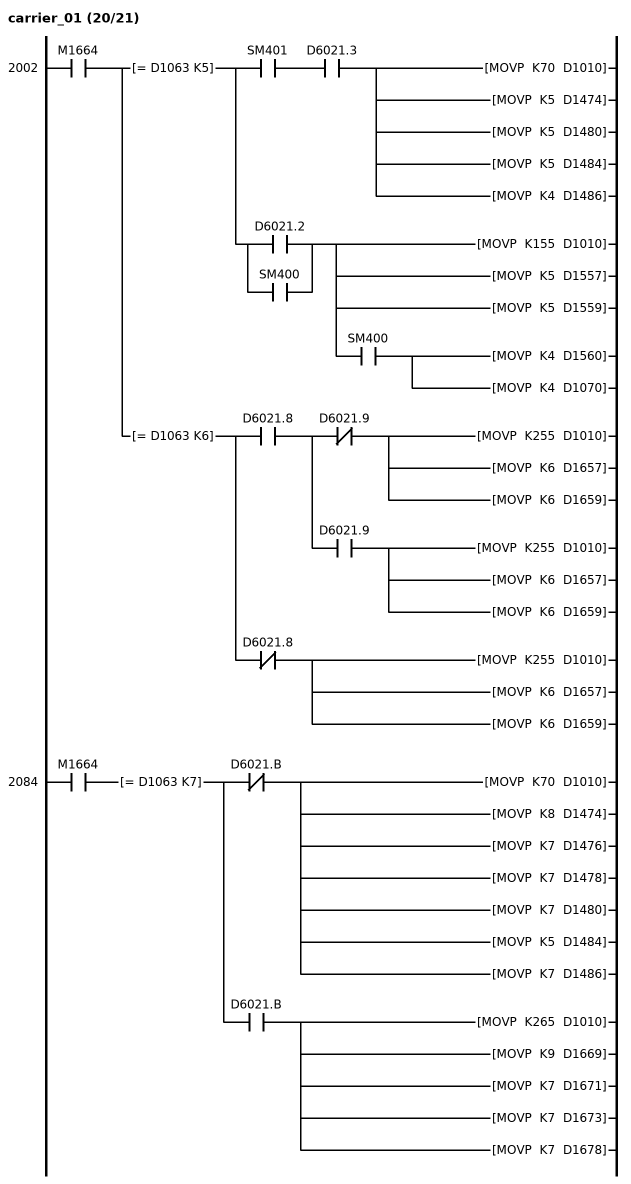
[picture p48: ladder of carrier_01, rungs at steps 2002 to 2084]
2002  LD      M1664
      MPS
      AND=    D1063 K5
      MPS
      AND     SM401
      AND     D6021.3
      MOVP    K70 D1010
      MOVP    K5 D1474
      MOVP    K5 D1480
      MOVP    K5 D1484
      MOVP    K4 D1486
      MPP
      LD      D6021.2
      OR      SM400
      ANB
      MOVP    K155 D1010
      MOVP    K5 D1557
      MOVP    K5 D1559
      AND     SM400
      MOVP    K4 D1560
      MOVP    K4 D1070
      MPP
      AND=    D1063 K6
      MPS
      AND     D6021.8
      MPS
      ANI     D6021.9
      MOVP    K255 D1010
      MOVP    K6 D1657
      MOVP    K6 D1659
      MPP
      AND     D6021.9
      MOVP    K255 D1010
      MOVP    K6 D1657
      MOVP    K6 D1659
      MPP
      ANI     D6021.8
      MOVP    K255 D1010
      MOVP    K6 D1657
      MOVP    K6 D1659
2084  LD      M1664
      AND=    D1063 K7
      MPS
      ANI     D6021.B
      MOVP    K70 D1010
      MOVP    K8 D1474
      MOVP    K7 D1476
      MOVP    K7 D1478
      MOVP    K7 D1480
      MOVP    K5 D1484
      MOVP    K7 D1486
      MPP
      AND     D6021.B
      MOVP    K265 D1010
      MOVP    K9 D1669
      MOVP    K7 D1671
      MOVP    K7 D1673
      MOVP    K7 D1678
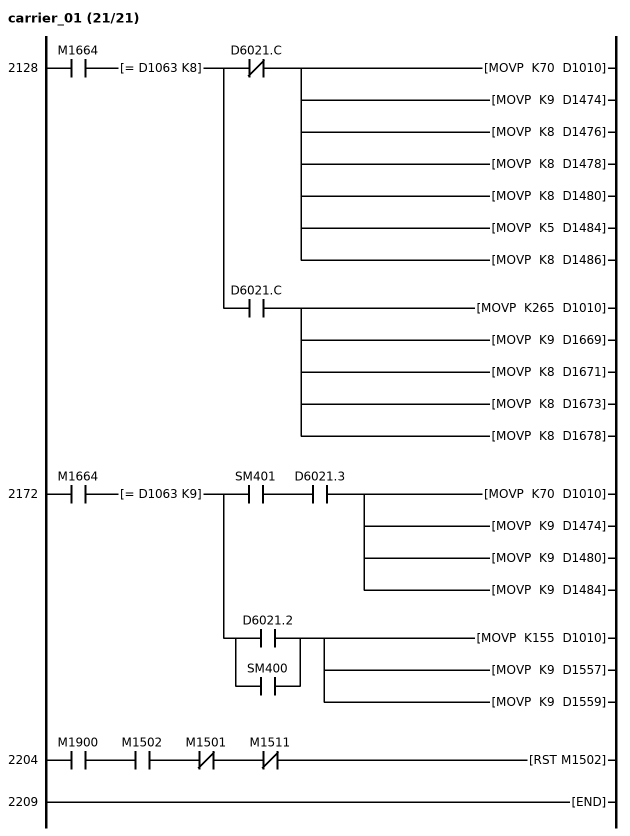
2128  LD      M1664
      AND=    D1063 K8
      MPS
      ANI     D6021.C
      MOVP    K70 D1010
      MOVP    K9 D1474
      MOVP    K8 D1476
      MOVP    K8 D1478
      MOVP    K8 D1480
      MOVP    K5 D1484
      MOVP    K8 D1486
      MPP
      AND     D6021.C
      MOVP    K265 D1010
      MOVP    K9 D1669
      MOVP    K8 D1671
      MOVP    K8 D1673
      MOVP    K8 D1678
2172  LD      M1664
      AND=    D1063 K9
      MPS
      AND     SM401
      AND     D6021.3
      MOVP    K70 D1010
      MOVP    K9 D1474
      MOVP    K9 D1480
      MOVP    K9 D1484
      MPP
      LD      D6021.2
      OR      SM400
      ANB
      MOVP    K155 D1010
      MOVP    K9 D1557
      MOVP    K9 D1559
2204  LD      M1900
      AND     M1502
      ANI     M1501
      ANI     M1511
      RST     M1502
2209  END
END_PROGRAM

PROGRAM carrier_02
VAR
  c_comm_2 : c_comm_2;
END_VAR
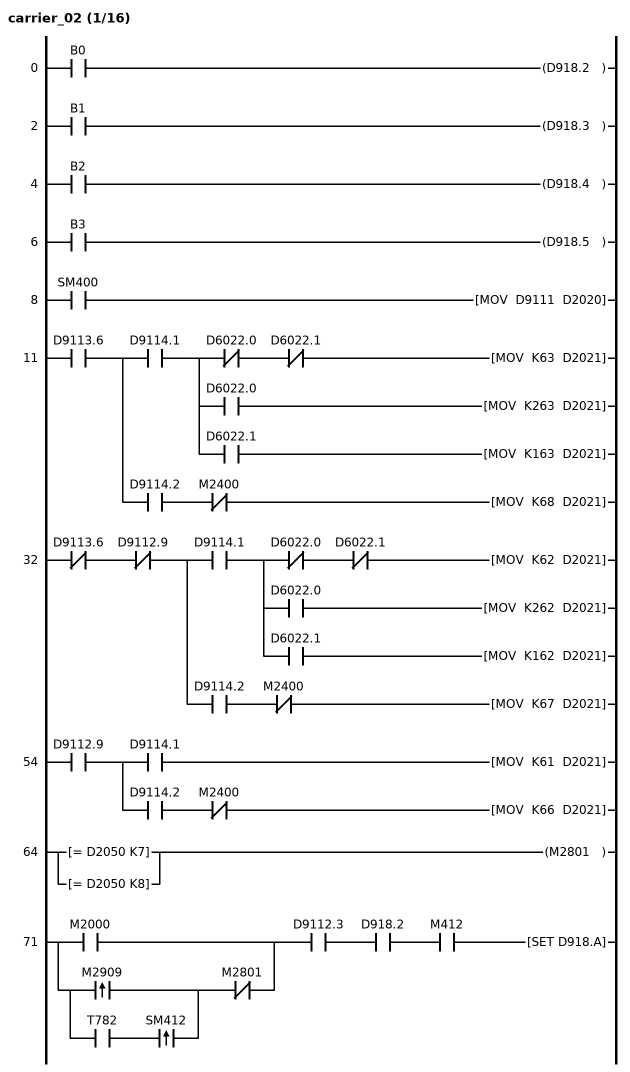
0     LD      B0
      OUT     D918.2
2     LD      B1
      OUT     D918.3
4     LD      B2
      OUT     D918.4
6     LD      B3
      OUT     D918.5
8     LD      SM400
      MOV     D9111 D2020
11    LD      D9113.6
      MPS
      AND     D9114.1
      MPS
      ANI     D6022.0
      ANI     D6022.1
      MOV     K63 D2021
      MRD
      AND     D6022.0
      MOV     K263 D2021
      MPP
      AND     D6022.1
      MOV     K163 D2021
      MPP
      AND     D9114.2
      ANI     M2400
      MOV     K68 D2021
32    LDI     D9113.6
      ANI     D9112.9
      MPS
      AND     D9114.1
      MPS
      ANI     D6022.0
      ANI     D6022.1
      MOV     K62 D2021
      MRD
      AND     D6022.0
      MOV     K262 D2021
      MPP
      AND     D6022.1
      MOV     K162 D2021
      MPP
      AND     D9114.2
      ANI     M2400
      MOV     K67 D2021
54    LD      D9112.9
      MPS
      AND     D9114.1
      MOV     K61 D2021
      MPP
      AND     D9114.2
      ANI     M2400
      MOV     K66 D2021
64    LD=     D2050 K7
      OR=     D2050 K8
      OUT     M2801
71    LD      M2000
      LDP     M2909
      LD      T782
      ANDP    SM412
      ORB
      ANI     M2801
      ORB
      AND     D9112.3
      AND     D918.2
      AND     M412
      SET     D918.A
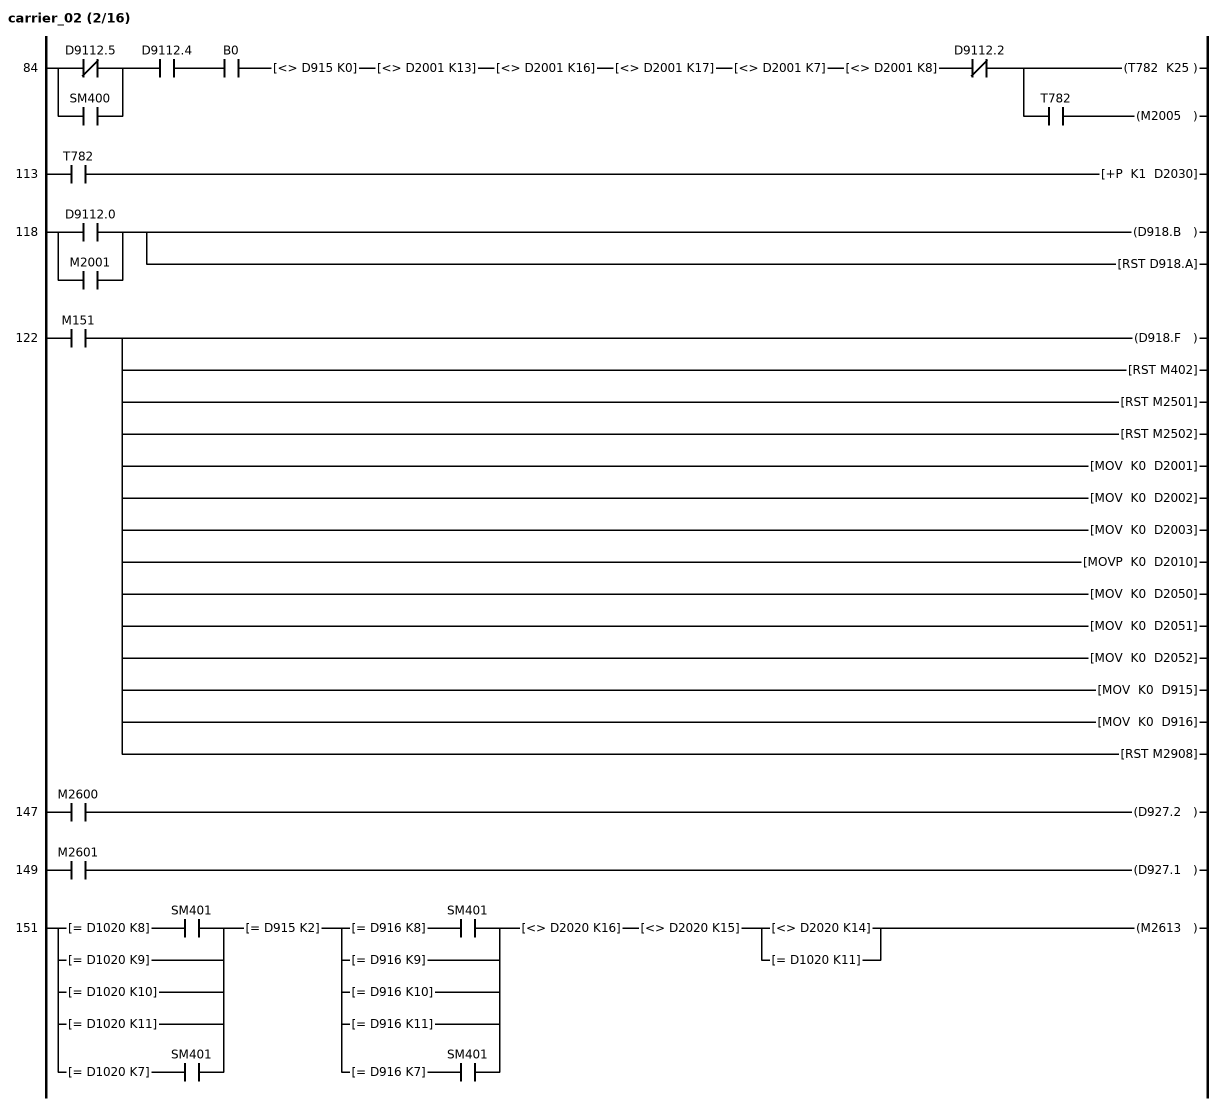
84    LDI     D9112.5
      OR      SM400
      AND     D9112.4
      AND     B0
      AND<>   D915 K0
      AND<>   D2001 K13
      AND<>   D2001 K16
      AND<>   D2001 K17
      AND<>   D2001 K7
      AND<>   D2001 K8
      ANI     D9112.2
      OUT     T782 K25
      AND     T782
      OUT     M2005
113   LD      T782
      +P      K1 D2030
118   LD      D9112.0
      OR      M2001
      OUT     D918.B
      RST     D918.A
122   LD      M151
      OUT     D918.F
      RST     M402
      RST     M2501
      RST     M2502
      MOV     K0 D2001
      MOV     K0 D2002
      MOV     K0 D2003
      MOVP    K0 D2010
      MOV     K0 D2050
      MOV     K0 D2051
      MOV     K0 D2052
      MOV     K0 D915
      MOV     K0 D916
      RST     M2908
147   LD      M2600
      OUT     D927.2
149   LD      M2601
      OUT     D927.1
151   LD=     D1020 K8
      AND     SM401
      OR=     D1020 K9
      OR=     D1020 K10
      OR=     D1020 K11
      LD=     D1020 K7
      AND     SM401
      ORB
      AND=    D915 K2
      LD=     D916 K8
      AND     SM401
      OR=     D916 K9
      OR=     D916 K10
      OR=     D916 K11
      LD=     D916 K7
      AND     SM401
      ORB
      ANB
      AND<>   D2020 K16
      AND<>   D2020 K15
      LD<>    D2020 K14
      OR=     D1020 K11
      ANB
      OUT     M2613
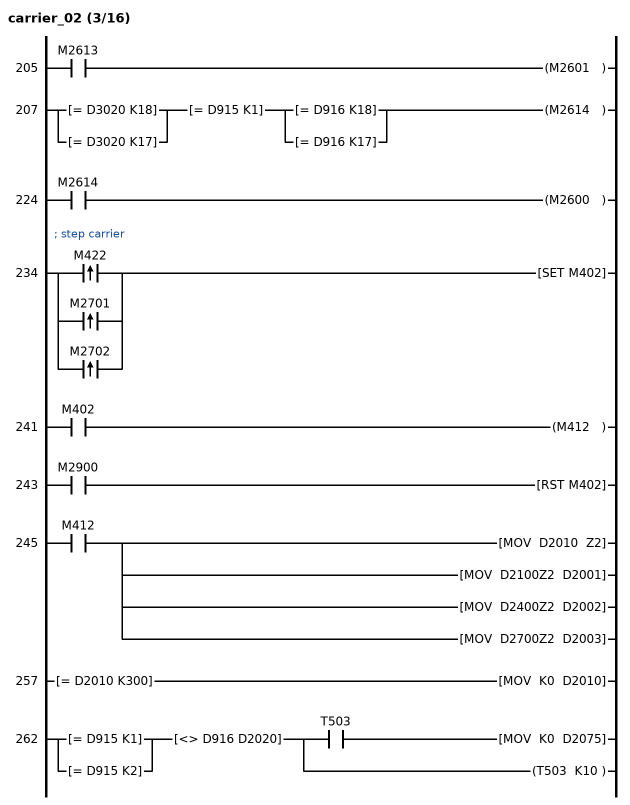
205   LD      M2613
      OUT     M2601
207   LD=     D3020 K18
      OR=     D3020 K17
      AND=    D915 K1
      LD=     D916 K18
      OR=     D916 K17
      ANB
      OUT     M2614
224   LD      M2614
      OUT     M2600
; step carrier
234   LDP     M422
      ORP     M2701
      ORP     M2702
      SET     M402
241   LD      M402
      OUT     M412
243   LD      M2900
      RST     M402
245   LD      M412
      MOV     D2010 Z2
      MOV     D2100Z2 D2001
      MOV     D2400Z2 D2002
      MOV     D2700Z2 D2003
257   LD=     D2010 K300
      MOV     K0 D2010
262   LD=     D915 K1
      OR=     D915 K2
      AND<>   D916 D2020
      MPS
      AND     T503
      MOV     K0 D2075
      MPP
      OUT     T503 K10
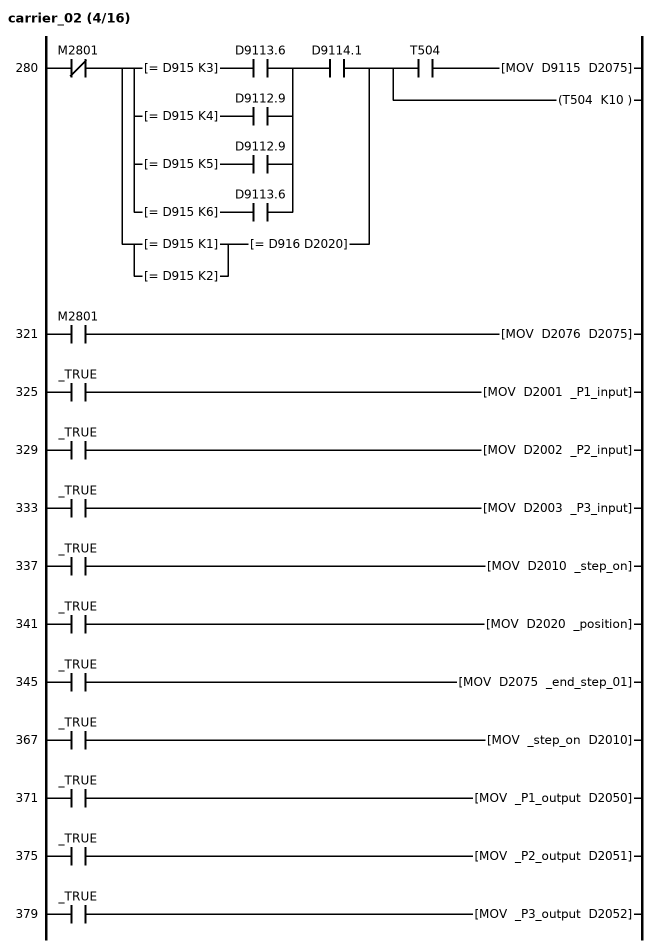
280   LDI     M2801
      LD=     D915 K3
      AND     D9113.6
      LD=     D915 K4
      AND     D9112.9
      ORB
      LD=     D915 K5
      AND     D9112.9
      ORB
      LD=     D915 K6
      AND     D9113.6
      ORB
      AND     D9114.1
      LD=     D915 K1
      OR=     D915 K2
      AND=    D916 D2020
      ORB
      ANB
      MPS
      AND     T504
      MOV     D9115 D2075
      MPP
      OUT     T504 K10
321   LD      M2801
      MOV     D2076 D2075
; FB BLK START c_comm_2(c_comm_2)
325   LD      _TRUE
      MOV     D2001 _P1_input
329   LD      _TRUE
      MOV     D2002 _P2_input
333   LD      _TRUE
      MOV     D2003 _P3_input
337   LD      _TRUE
      MOV     D2010 _step_on
341   LD      _TRUE
      MOV     D2020 _position
345   LD      _TRUE
      MOV     D2075 _end_step_01
; FB START
; FB_NAME c_comm_2
; INSTANCE_NAME c_comm_2
; FB IN_W:P1_input
; FB OUT_step_on:W
; FB IN_W:P2_input
; FB OUT_P1_output:W
; FB IN_W:P3_input
; FB OUT_P2_output:W
; FB IN_W:step_on
; FB OUT_P3_output:W
; FB IN_W:position
; FB OUT_end_step_01:W
; FB IN_W:end_step_01
; FB OUT_end_signal:B
; FB OUT_next_signal:B
; FB OUT_punch:B
; FB END
367   LD      _TRUE
      MOV     _step_on D2010
371   LD      _TRUE
      MOV     _P1_output D2050
375   LD      _TRUE
      MOV     _P2_output D2051
379   LD      _TRUE
      MOV     _P3_output D2052
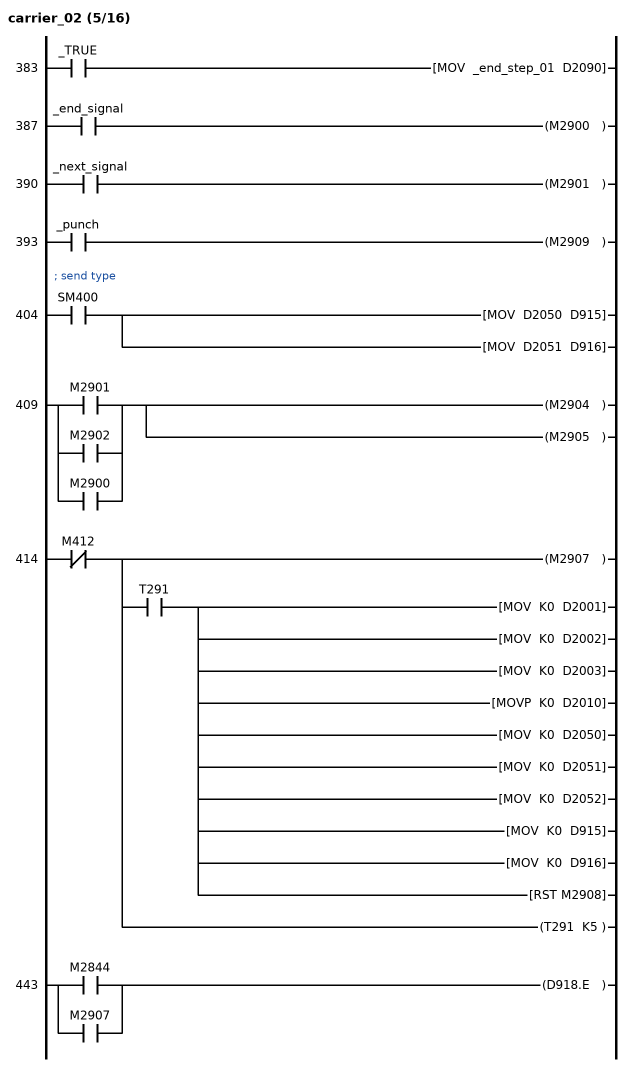
383   LD      _TRUE
      MOV     _end_step_01 D2090
387   LD      _end_signal
      OUT     M2900
390   LD      _next_signal
      OUT     M2901
393   LD      _punch
      OUT     M2909
; FB BLK END
; send type
404   LD      SM400
      MOV     D2050 D915
      MOV     D2051 D916
409   LD      M2901
      OR      M2902
      OR      M2900
      OUT     M2904
      OUT     M2905
414   LDI     M412
      OUT     M2907
      MPS
      AND     T291
      MOV     K0 D2001
      MOV     K0 D2002
      MOV     K0 D2003
      MOVP    K0 D2010
      MOV     K0 D2050
      MOV     K0 D2051
      MOV     K0 D2052
      MOV     K0 D915
      MOV     K0 D916
      RST     M2908
      MPP
      OUT     T291 K5
443   LD      M2844
      OR      M2907
      OUT     D918.E
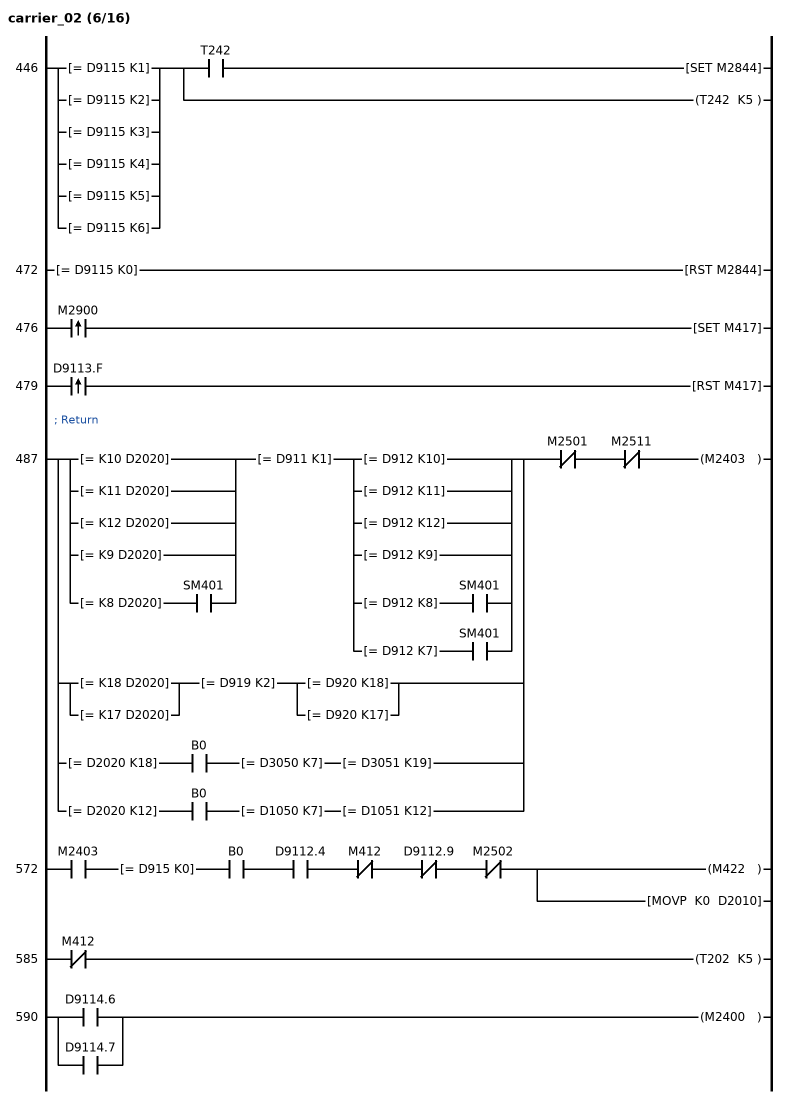
446   LD=     D9115 K1
      OR=     D9115 K2
      OR=     D9115 K3
      OR=     D9115 K4
      OR=     D9115 K5
      OR=     D9115 K6
      MPS
      AND     T242
      SET     M2844
      MPP
      OUT     T242 K5
472   LD=     D9115 K0
      RST     M2844
476   LDP     M2900
      SET     M417
479   LDP     D9113.F
      RST     M417
; Return
487   LD=     K10 D2020
      OR=     K11 D2020
      OR=     K12 D2020
      OR=     K9 D2020
      LD=     K8 D2020
      AND     SM401
      ORB
      AND=    D911 K1
      LD=     D912 K10
      OR=     D912 K11
      OR=     D912 K12
      OR=     D912 K9
      LD=     D912 K8
      AND     SM401
      ORB
      LD=     D912 K7
      AND     SM401
      ORB
      ANB
      LD=     K18 D2020
      OR=     K17 D2020
      AND=    D919 K2
      LD=     D920 K18
      OR=     D920 K17
      ANB
      ORB
      LD=     D2020 K18
      AND     B0
      AND=    D3050 K7
      AND=    D3051 K19
      ORB
      LD=     D2020 K12
      AND     B0
      AND=    D1050 K7
      AND=    D1051 K12
      ORB
      ANI     M2501
      ANI     M2511
      OUT     M2403
572   LD      M2403
      AND=    D915 K0
      AND     B0
      AND     D9112.4
      ANI     M412
      ANI     D9112.9
      ANI     M2502
      OUT     M422
      MOVP    K0 D2010
585   LDI     M412
      OUT     T202 K5
590   LD      D9114.6
      OR      D9114.7
      OUT     M2400
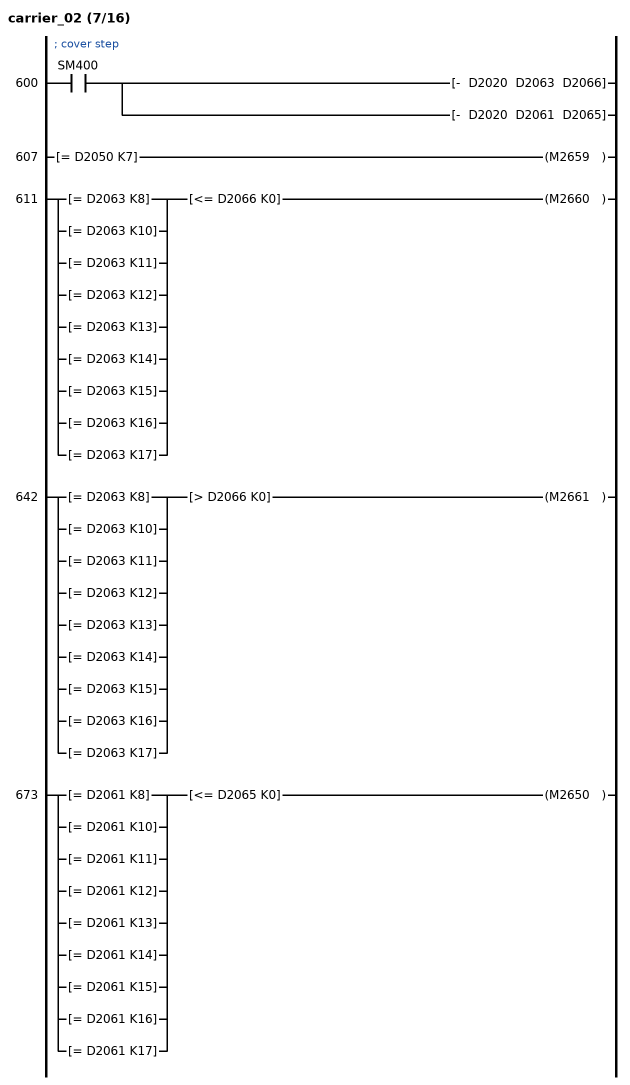
; cover step
600   LD      SM400
      -       D2020 D2063 D2066
      -       D2020 D2061 D2065
607   LD=     D2050 K7
      OUT     M2659
611   LD=     D2063 K8
      OR=     D2063 K10
      OR=     D2063 K11
      OR=     D2063 K12
      OR=     D2063 K13
      OR=     D2063 K14
      OR=     D2063 K15
      OR=     D2063 K16
      OR=     D2063 K17
      AND<=   D2066 K0
      OUT     M2660
642   LD=     D2063 K8
      OR=     D2063 K10
      OR=     D2063 K11
      OR=     D2063 K12
      OR=     D2063 K13
      OR=     D2063 K14
      OR=     D2063 K15
      OR=     D2063 K16
      OR=     D2063 K17
      AND>    D2066 K0
      OUT     M2661
673   LD=     D2061 K8
      OR=     D2061 K10
      OR=     D2061 K11
      OR=     D2061 K12
      OR=     D2061 K13
      OR=     D2061 K14
      OR=     D2061 K15
      OR=     D2061 K16
      OR=     D2061 K17
      AND<=   D2065 K0
      OUT     M2650
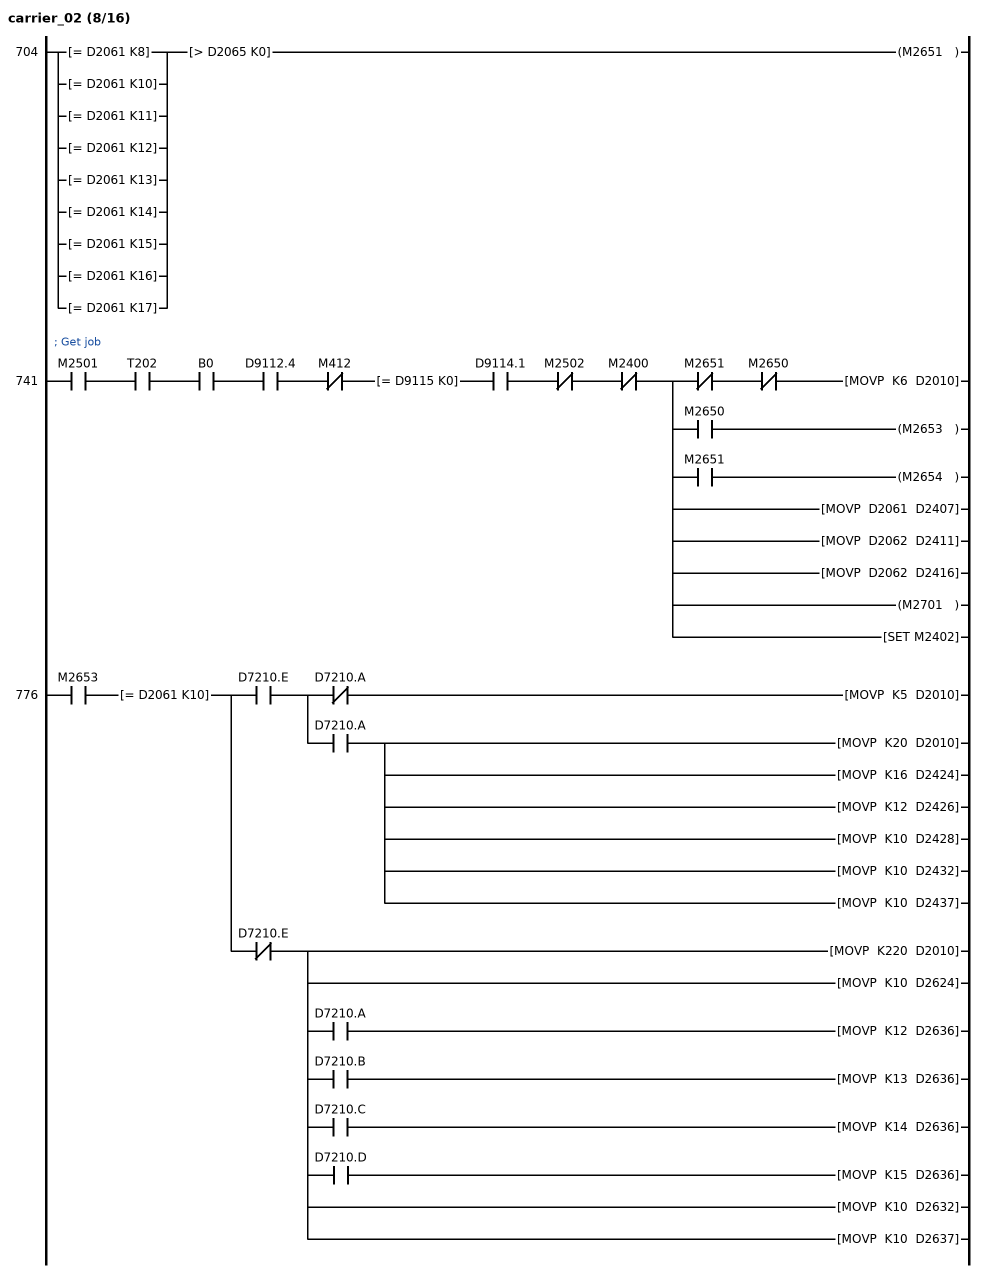
704   LD=     D2061 K8
      OR=     D2061 K10
      OR=     D2061 K11
      OR=     D2061 K12
      OR=     D2061 K13
      OR=     D2061 K14
      OR=     D2061 K15
      OR=     D2061 K16
      OR=     D2061 K17
      AND>    D2065 K0
      OUT     M2651
; Get job
741   LD      M2501
      AND     T202
      AND     B0
      AND     D9112.4
      ANI     M412
      AND=    D9115 K0
      AND     D9114.1
      ANI     M2502
      ANI     M2400
      MPS
      ANI     M2651
      ANI     M2650
      MOVP    K6 D2010
      MRD
      AND     M2650
      OUT     M2653
      MRD
      AND     M2651
      OUT     M2654
      MPP
      MOVP    D2061 D2407
      MOVP    D2062 D2411
      MOVP    D2062 D2416
      OUT     M2701
      SET     M2402
776   LD      M2653
      AND=    D2061 K10
      MPS
      AND     D7210.E
      MPS
      ANI     D7210.A
      MOVP    K5 D2010
      MPP
      AND     D7210.A
      MOVP    K20 D2010
      MOVP    K16 D2424
      MOVP    K12 D2426
      MOVP    K10 D2428
      MOVP    K10 D2432
      MOVP    K10 D2437
      MPP
      ANI     D7210.E
      MOVP    K220 D2010
      MOVP    K10 D2624
      MPS
      AND     D7210.A
      MOVP    K12 D2636
      MRD
      AND     D7210.B
      MOVP    K13 D2636
      MRD
      AND     D7210.C
      MOVP    K14 D2636
      MRD
      AND     D7210.D
      MOVP    K15 D2636
      MPP
      MOVP    K10 D2632
      MOVP    K10 D2637
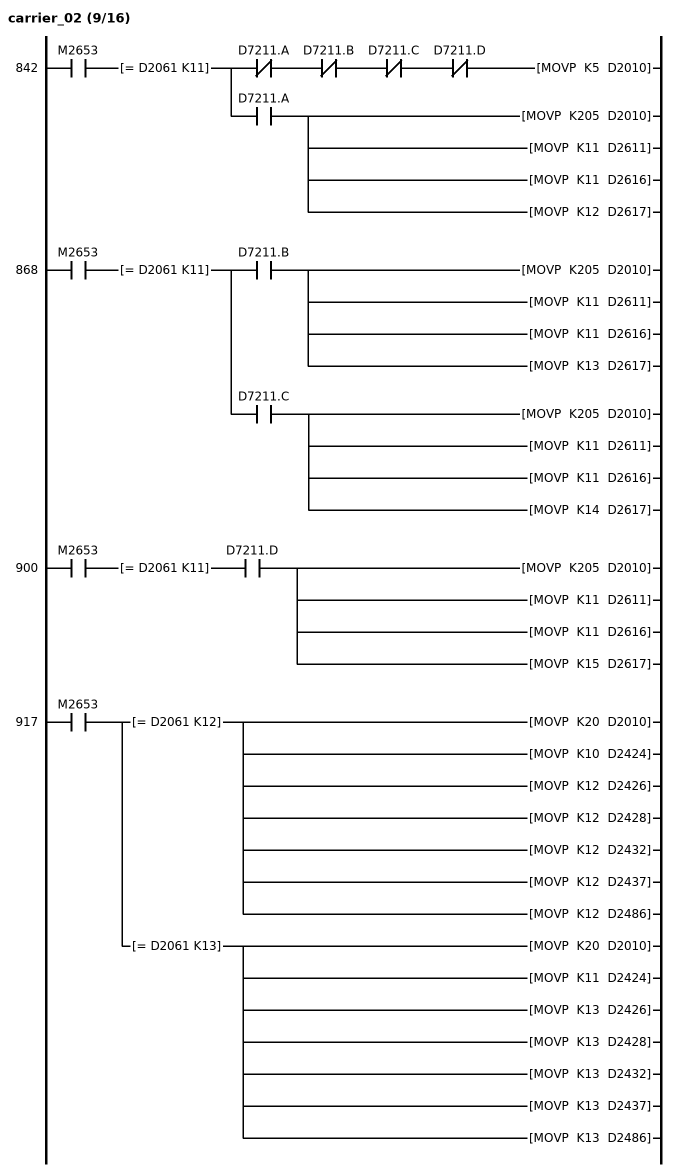
842   LD      M2653
      AND=    D2061 K11
      MPS
      ANI     D7211.A
      ANI     D7211.B
      ANI     D7211.C
      ANI     D7211.D
      MOVP    K5 D2010
      MPP
      AND     D7211.A
      MOVP    K205 D2010
      MOVP    K11 D2611
      MOVP    K11 D2616
      MOVP    K12 D2617
868   LD      M2653
      AND=    D2061 K11
      MPS
      AND     D7211.B
      MOVP    K205 D2010
      MOVP    K11 D2611
      MOVP    K11 D2616
      MOVP    K13 D2617
      MPP
      AND     D7211.C
      MOVP    K205 D2010
      MOVP    K11 D2611
      MOVP    K11 D2616
      MOVP    K14 D2617
900   LD      M2653
      AND=    D2061 K11
      AND     D7211.D
      MOVP    K205 D2010
      MOVP    K11 D2611
      MOVP    K11 D2616
      MOVP    K15 D2617
917   LD      M2653
      MPS
      AND=    D2061 K12
      MOVP    K20 D2010
      MOVP    K10 D2424
      MOVP    K12 D2426
      MOVP    K12 D2428
      MOVP    K12 D2432
      MOVP    K12 D2437
      MOVP    K12 D2486
      MPP
      AND=    D2061 K13
      MOVP    K20 D2010
      MOVP    K11 D2424
      MOVP    K13 D2426
      MOVP    K13 D2428
      MOVP    K13 D2432
      MOVP    K13 D2437
      MOVP    K13 D2486
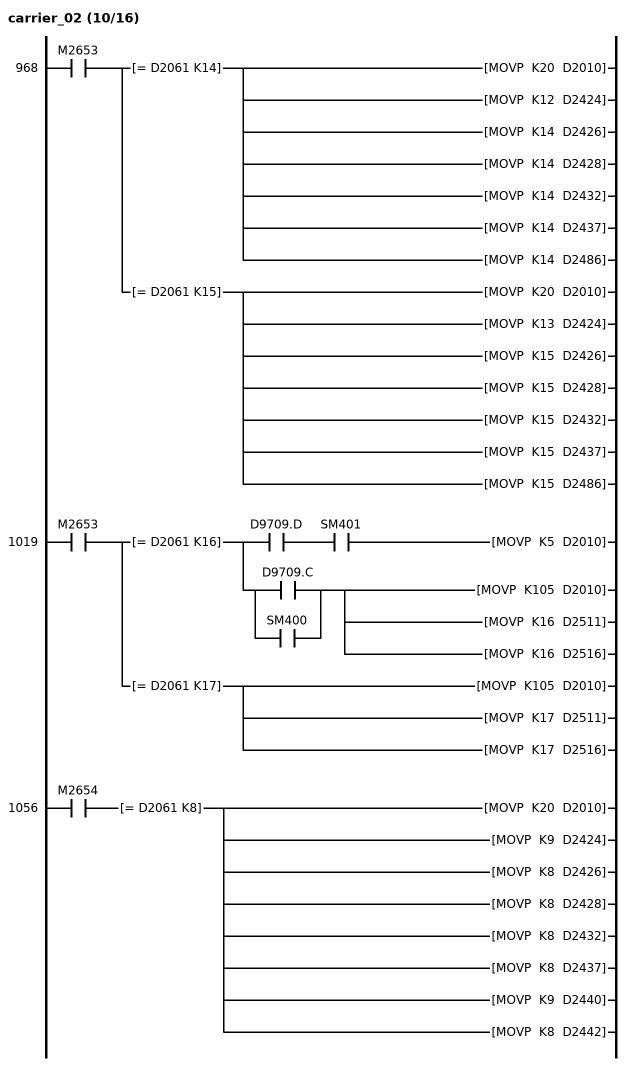
968   LD      M2653
      MPS
      AND=    D2061 K14
      MOVP    K20 D2010
      MOVP    K12 D2424
      MOVP    K14 D2426
      MOVP    K14 D2428
      MOVP    K14 D2432
      MOVP    K14 D2437
      MOVP    K14 D2486
      MPP
      AND=    D2061 K15
      MOVP    K20 D2010
      MOVP    K13 D2424
      MOVP    K15 D2426
      MOVP    K15 D2428
      MOVP    K15 D2432
      MOVP    K15 D2437
      MOVP    K15 D2486
1019  LD      M2653
      MPS
      AND=    D2061 K16
      MPS
      AND     D9709.D
      AND     SM401
      MOVP    K5 D2010
      MPP
      LD      D9709.C
      OR      SM400
      ANB
      MOVP    K105 D2010
      MOVP    K16 D2511
      MOVP    K16 D2516
      MPP
      AND=    D2061 K17
      MOVP    K105 D2010
      MOVP    K17 D2511
      MOVP    K17 D2516
1056  LD      M2654
      AND=    D2061 K8
      MOVP    K20 D2010
      MOVP    K9 D2424
      MOVP    K8 D2426
      MOVP    K8 D2428
      MOVP    K8 D2432
      MOVP    K8 D2437
      MOVP    K9 D2440
      MOVP    K8 D2442
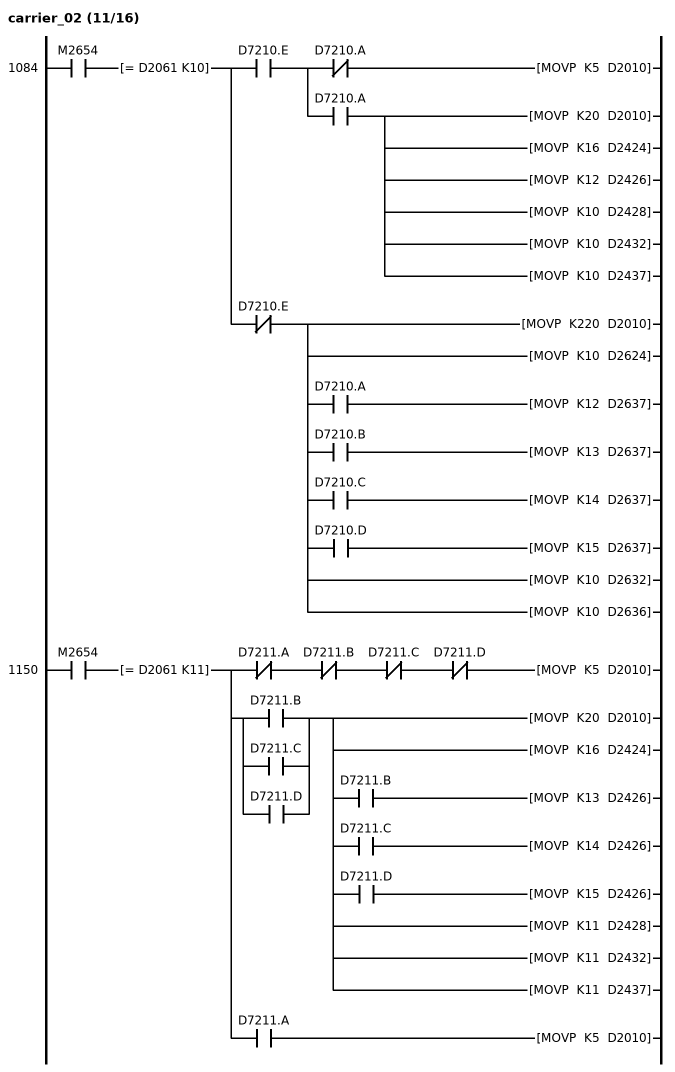
1084  LD      M2654
      AND=    D2061 K10
      MPS
      AND     D7210.E
      MPS
      ANI     D7210.A
      MOVP    K5 D2010
      MPP
      AND     D7210.A
      MOVP    K20 D2010
      MOVP    K16 D2424
      MOVP    K12 D2426
      MOVP    K10 D2428
      MOVP    K10 D2432
      MOVP    K10 D2437
      MPP
      ANI     D7210.E
      MOVP    K220 D2010
      MOVP    K10 D2624
      MPS
      AND     D7210.A
      MOVP    K12 D2637
      MRD
      AND     D7210.B
      MOVP    K13 D2637
      MRD
      AND     D7210.C
      MOVP    K14 D2637
      MRD
      AND     D7210.D
      MOVP    K15 D2637
      MPP
      MOVP    K10 D2632
      MOVP    K10 D2636
1150  LD      M2654
      AND=    D2061 K11
      MPS
      ANI     D7211.A
      ANI     D7211.B
      ANI     D7211.C
      ANI     D7211.D
      MOVP    K5 D2010
      MRD
      LD      D7211.B
      OR      D7211.C
      OR      D7211.D
      ANB
      MOVP    K20 D2010
      MOVP    K16 D2424
      MPS
      AND     D7211.B
      MOVP    K13 D2426
      MRD
      AND     D7211.C
      MOVP    K14 D2426
      MRD
      AND     D7211.D
      MOVP    K15 D2426
      MPP
      MOVP    K11 D2428
      MOVP    K11 D2432
      MOVP    K11 D2437
      MPP
      AND     D7211.A
      MOVP    K5 D2010
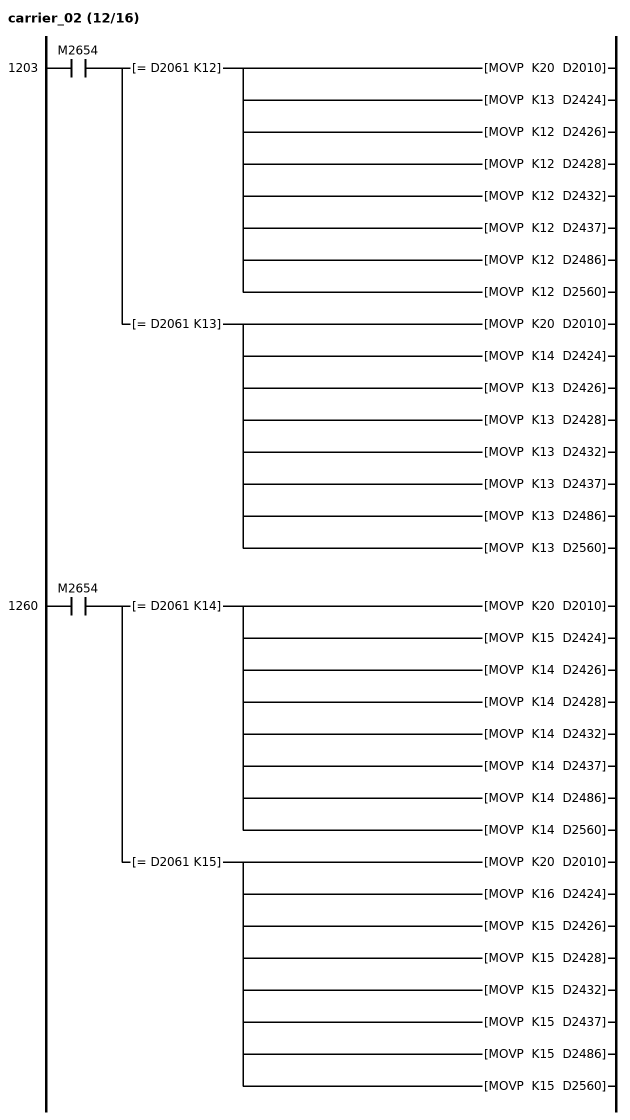
1203  LD      M2654
      MPS
      AND=    D2061 K12
      MOVP    K20 D2010
      MOVP    K13 D2424
      MOVP    K12 D2426
      MOVP    K12 D2428
      MOVP    K12 D2432
      MOVP    K12 D2437
      MOVP    K12 D2486
      MOVP    K12 D2560
      MPP
      AND=    D2061 K13
      MOVP    K20 D2010
      MOVP    K14 D2424
      MOVP    K13 D2426
      MOVP    K13 D2428
      MOVP    K13 D2432
      MOVP    K13 D2437
      MOVP    K13 D2486
      MOVP    K13 D2560
1260  LD      M2654
      MPS
      AND=    D2061 K14
      MOVP    K20 D2010
      MOVP    K15 D2424
      MOVP    K14 D2426
      MOVP    K14 D2428
      MOVP    K14 D2432
      MOVP    K14 D2437
      MOVP    K14 D2486
      MOVP    K14 D2560
      MPP
      AND=    D2061 K15
      MOVP    K20 D2010
      MOVP    K16 D2424
      MOVP    K15 D2426
      MOVP    K15 D2428
      MOVP    K15 D2432
      MOVP    K15 D2437
      MOVP    K15 D2486
      MOVP    K15 D2560
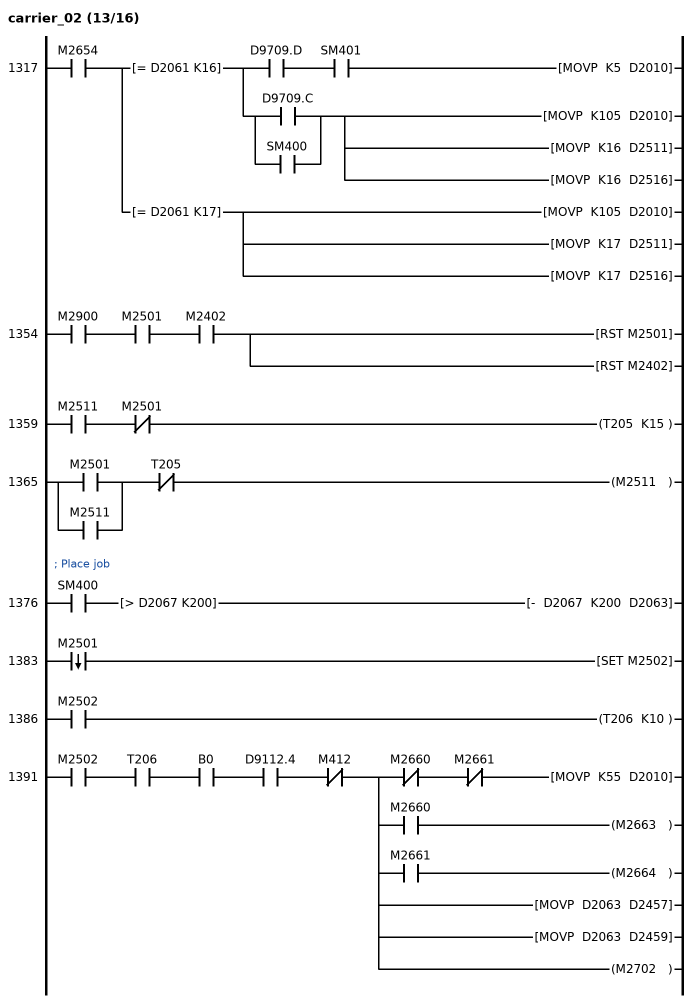
1317  LD      M2654
      MPS
      AND=    D2061 K16
      MPS
      AND     D9709.D
      AND     SM401
      MOVP    K5 D2010
      MPP
      LD      D9709.C
      OR      SM400
      ANB
      MOVP    K105 D2010
      MOVP    K16 D2511
      MOVP    K16 D2516
      MPP
      AND=    D2061 K17
      MOVP    K105 D2010
      MOVP    K17 D2511
      MOVP    K17 D2516
1354  LD      M2900
      AND     M2501
      AND     M2402
      RST     M2501
      RST     M2402
1359  LD      M2511
      ANI     M2501
      OUT     T205 K15
1365  LD      M2501
      OR      M2511
      ANI     T205
      OUT     M2511
; Place job
1376  LD      SM400
      AND>    D2067 K200
      -       D2067 K200 D2063
1383  LDF     M2501
      SET     M2502
1386  LD      M2502
      OUT     T206 K10
1391  LD      M2502
      AND     T206
      AND     B0
      AND     D9112.4
      ANI     M412
      MPS
      ANI     M2660
      ANI     M2661
      MOVP    K55 D2010
      MRD
      AND     M2660
      OUT     M2663
      MRD
      AND     M2661
      OUT     M2664
      MPP
      MOVP    D2063 D2457
      MOVP    D2063 D2459
      OUT     M2702
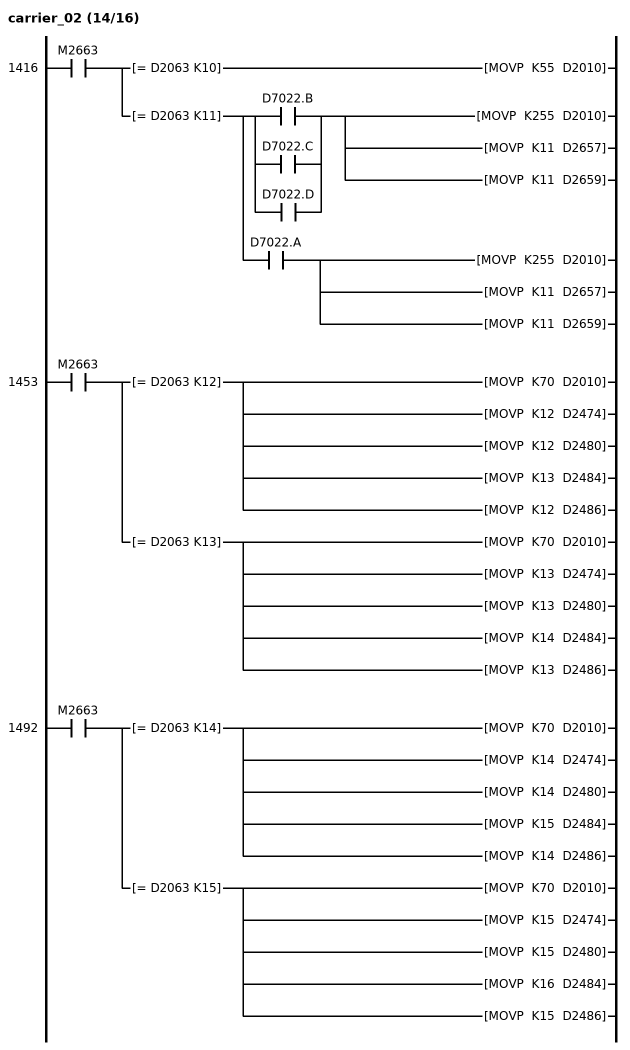
1416  LD      M2663
      MPS
      AND=    D2063 K10
      MOVP    K55 D2010
      MPP
      AND=    D2063 K11
      MPS
      LD      D7022.B
      OR      D7022.C
      OR      D7022.D
      ANB
      MOVP    K255 D2010
      MOVP    K11 D2657
      MOVP    K11 D2659
      MPP
      AND     D7022.A
      MOVP    K255 D2010
      MOVP    K11 D2657
      MOVP    K11 D2659
1453  LD      M2663
      MPS
      AND=    D2063 K12
      MOVP    K70 D2010
      MOVP    K12 D2474
      MOVP    K12 D2480
      MOVP    K13 D2484
      MOVP    K12 D2486
      MPP
      AND=    D2063 K13
      MOVP    K70 D2010
      MOVP    K13 D2474
      MOVP    K13 D2480
      MOVP    K14 D2484
      MOVP    K13 D2486
1492  LD      M2663
      MPS
      AND=    D2063 K14
      MOVP    K70 D2010
      MOVP    K14 D2474
      MOVP    K14 D2480
      MOVP    K15 D2484
      MOVP    K14 D2486
      MPP
      AND=    D2063 K15
      MOVP    K70 D2010
      MOVP    K15 D2474
      MOVP    K15 D2480
      MOVP    K16 D2484
      MOVP    K15 D2486
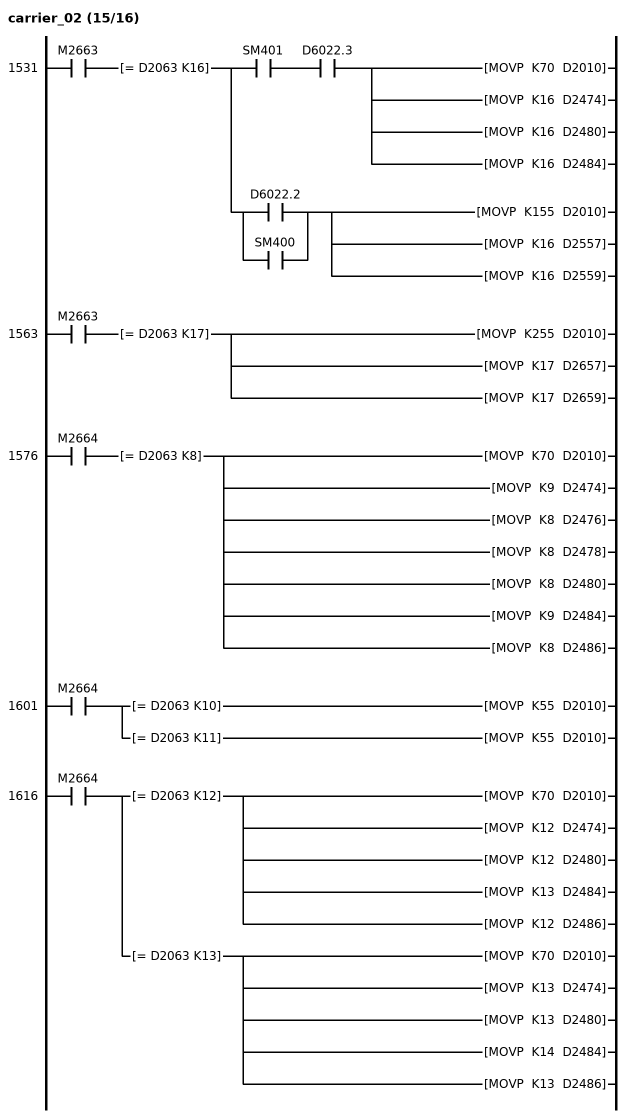
1531  LD      M2663
      AND=    D2063 K16
      MPS
      AND     SM401
      AND     D6022.3
      MOVP    K70 D2010
      MOVP    K16 D2474
      MOVP    K16 D2480
      MOVP    K16 D2484
      MPP
      LD      D6022.2
      OR      SM400
      ANB
      MOVP    K155 D2010
      MOVP    K16 D2557
      MOVP    K16 D2559
1563  LD      M2663
      AND=    D2063 K17
      MOVP    K255 D2010
      MOVP    K17 D2657
      MOVP    K17 D2659
1576  LD      M2664
      AND=    D2063 K8
      MOVP    K70 D2010
      MOVP    K9 D2474
      MOVP    K8 D2476
      MOVP    K8 D2478
      MOVP    K8 D2480
      MOVP    K9 D2484
      MOVP    K8 D2486
1601  LD      M2664
      MPS
      AND=    D2063 K10
      MOVP    K55 D2010
      MPP
      AND=    D2063 K11
      MOVP    K55 D2010
1616  LD      M2664
      MPS
      AND=    D2063 K12
      MOVP    K70 D2010
      MOVP    K12 D2474
      MOVP    K12 D2480
      MOVP    K13 D2484
      MOVP    K12 D2486
      MPP
      AND=    D2063 K13
      MOVP    K70 D2010
      MOVP    K13 D2474
      MOVP    K13 D2480
      MOVP    K14 D2484
      MOVP    K13 D2486
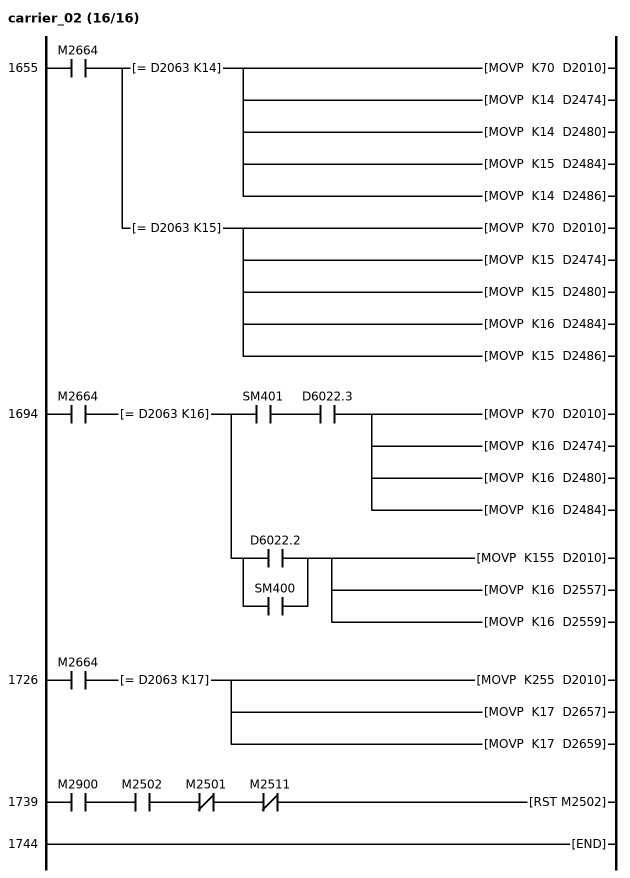
1655  LD      M2664
      MPS
      AND=    D2063 K14
      MOVP    K70 D2010
      MOVP    K14 D2474
      MOVP    K14 D2480
      MOVP    K15 D2484
      MOVP    K14 D2486
      MPP
      AND=    D2063 K15
      MOVP    K70 D2010
      MOVP    K15 D2474
      MOVP    K15 D2480
      MOVP    K16 D2484
      MOVP    K15 D2486
1694  LD      M2664
      AND=    D2063 K16
      MPS
      AND     SM401
      AND     D6022.3
      MOVP    K70 D2010
      MOVP    K16 D2474
      MOVP    K16 D2480
      MOVP    K16 D2484
      MPP
      LD      D6022.2
      OR      SM400
      ANB
      MOVP    K155 D2010
      MOVP    K16 D2557
      MOVP    K16 D2559
1726  LD      M2664
      AND=    D2063 K17
      MOVP    K255 D2010
      MOVP    K17 D2657
      MOVP    K17 D2659
1739  LD      M2900
      AND     M2502
      ANI     M2501
      ANI     M2511
      RST     M2502
1744  END
END_PROGRAM

PROGRAM carrier_03
VAR
  c_comm_3 : c_comm_3;
END_VAR
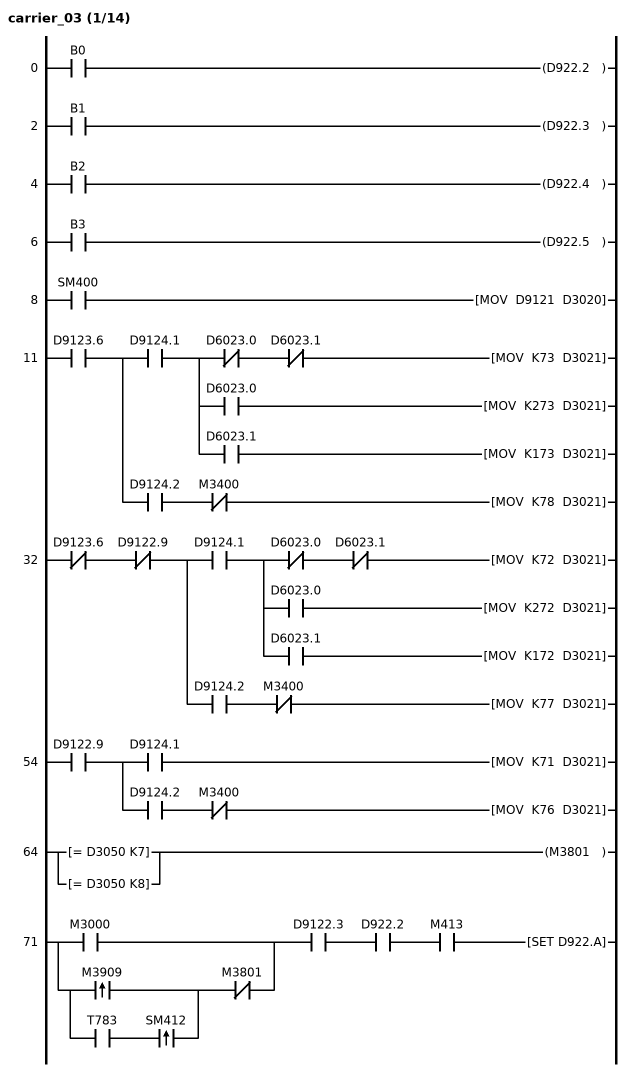
0     LD      B0
      OUT     D922.2
2     LD      B1
      OUT     D922.3
4     LD      B2
      OUT     D922.4
6     LD      B3
      OUT     D922.5
8     LD      SM400
      MOV     D9121 D3020
11    LD      D9123.6
      MPS
      AND     D9124.1
      MPS
      ANI     D6023.0
      ANI     D6023.1
      MOV     K73 D3021
      MRD
      AND     D6023.0
      MOV     K273 D3021
      MPP
      AND     D6023.1
      MOV     K173 D3021
      MPP
      AND     D9124.2
      ANI     M3400
      MOV     K78 D3021
32    LDI     D9123.6
      ANI     D9122.9
      MPS
      AND     D9124.1
      MPS
      ANI     D6023.0
      ANI     D6023.1
      MOV     K72 D3021
      MRD
      AND     D6023.0
      MOV     K272 D3021
      MPP
      AND     D6023.1
      MOV     K172 D3021
      MPP
      AND     D9124.2
      ANI     M3400
      MOV     K77 D3021
54    LD      D9122.9
      MPS
      AND     D9124.1
      MOV     K71 D3021
      MPP
      AND     D9124.2
      ANI     M3400
      MOV     K76 D3021
64    LD=     D3050 K7
      OR=     D3050 K8
      OUT     M3801
71    LD      M3000
      LDP     M3909
      LD      T783
      ANDP    SM412
      ORB
      ANI     M3801
      ORB
      AND     D9122.3
      AND     D922.2
      AND     M413
      SET     D922.A
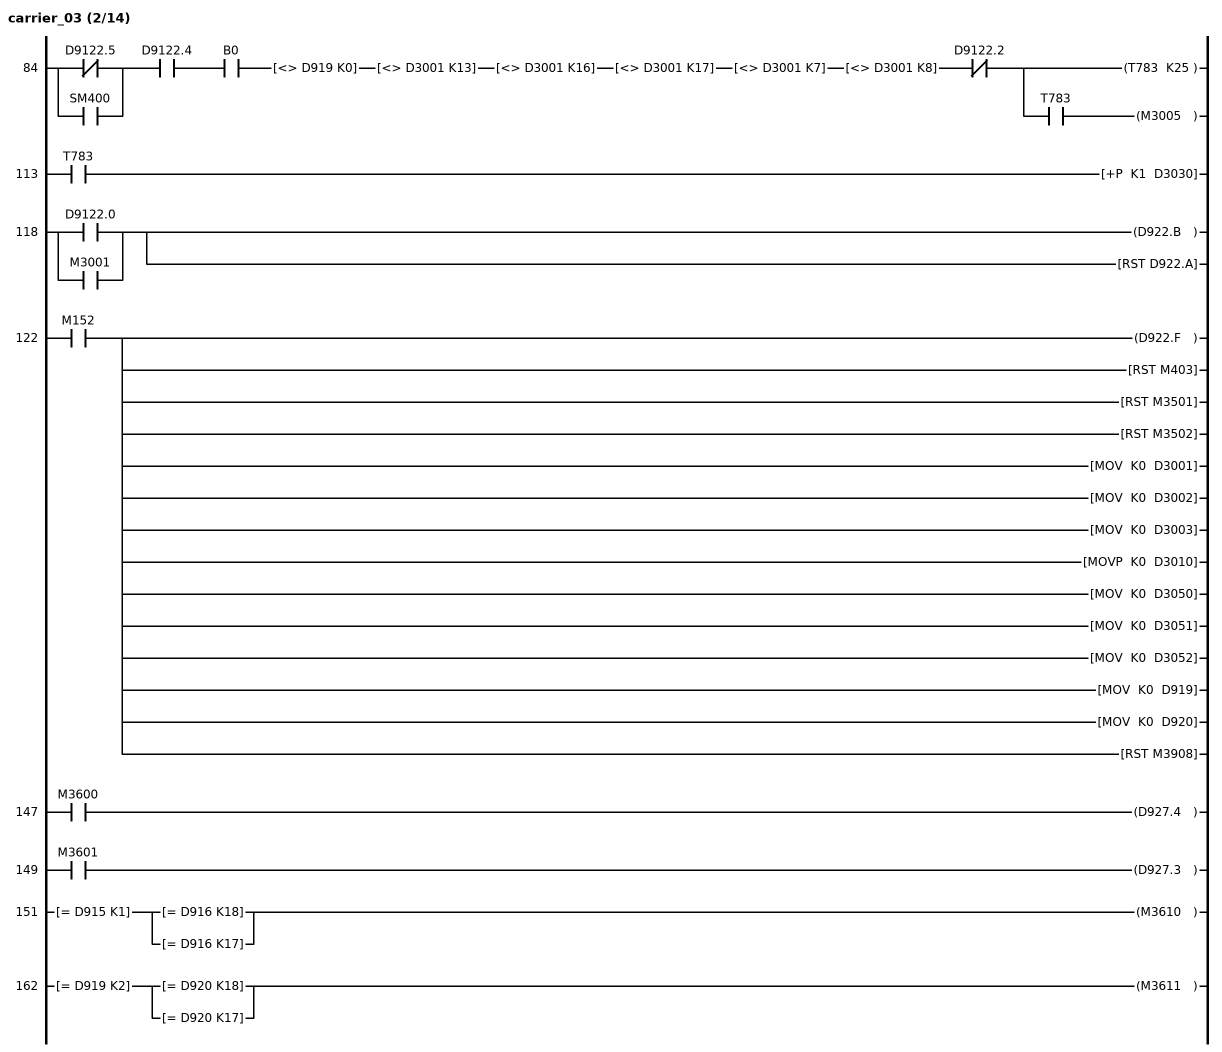
84    LDI     D9122.5
      OR      SM400
      AND     D9122.4
      AND     B0
      AND<>   D919 K0
      AND<>   D3001 K13
      AND<>   D3001 K16
      AND<>   D3001 K17
      AND<>   D3001 K7
      AND<>   D3001 K8
      ANI     D9122.2
      OUT     T783 K25
      AND     T783
      OUT     M3005
113   LD      T783
      +P      K1 D3030
118   LD      D9122.0
      OR      M3001
      OUT     D922.B
      RST     D922.A
122   LD      M152
      OUT     D922.F
      RST     M403
      RST     M3501
      RST     M3502
      MOV     K0 D3001
      MOV     K0 D3002
      MOV     K0 D3003
      MOVP    K0 D3010
      MOV     K0 D3050
      MOV     K0 D3051
      MOV     K0 D3052
      MOV     K0 D919
      MOV     K0 D920
      RST     M3908
147   LD      M3600
      OUT     D927.4
149   LD      M3601
      OUT     D927.3
151   LD=     D915 K1
      LD=     D916 K18
      OR=     D916 K17
      ANB
      OUT     M3610
162   LD=     D919 K2
      LD=     D920 K18
      OR=     D920 K17
      ANB
      OUT     M3611
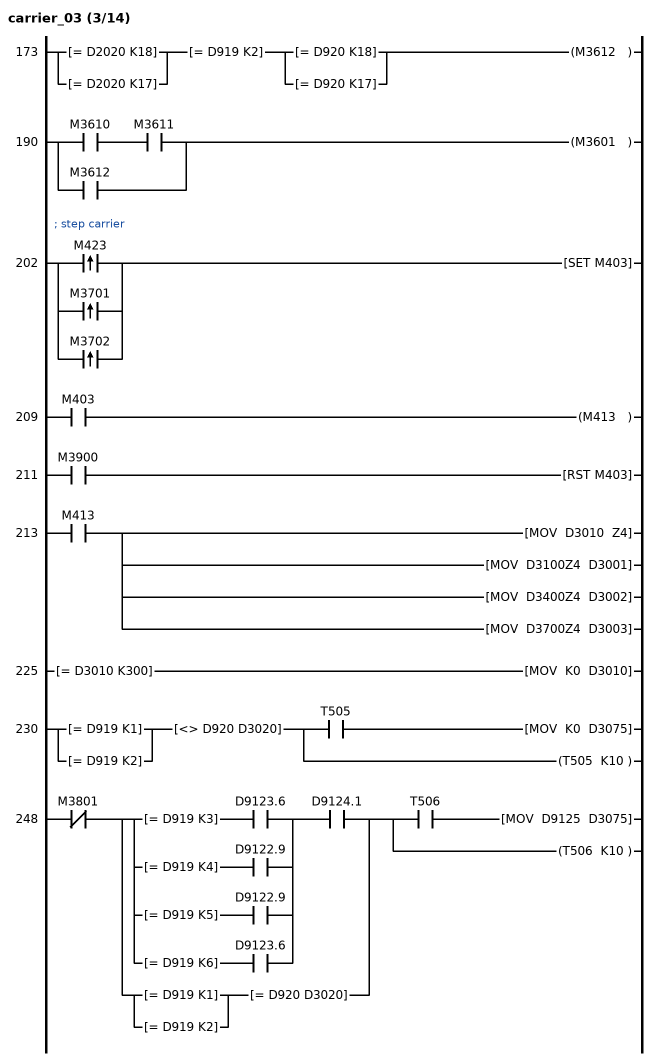
173   LD=     D2020 K18
      OR=     D2020 K17
      AND=    D919 K2
      LD=     D920 K18
      OR=     D920 K17
      ANB
      OUT     M3612
190   LD      M3610
      AND     M3611
      OR      M3612
      OUT     M3601
; step carrier
202   LDP     M423
      ORP     M3701
      ORP     M3702
      SET     M403
209   LD      M403
      OUT     M413
211   LD      M3900
      RST     M403
213   LD      M413
      MOV     D3010 Z4
      MOV     D3100Z4 D3001
      MOV     D3400Z4 D3002
      MOV     D3700Z4 D3003
225   LD=     D3010 K300
      MOV     K0 D3010
230   LD=     D919 K1
      OR=     D919 K2
      AND<>   D920 D3020
      MPS
      AND     T505
      MOV     K0 D3075
      MPP
      OUT     T505 K10
248   LDI     M3801
      LD=     D919 K3
      AND     D9123.6
      LD=     D919 K4
      AND     D9122.9
      ORB
      LD=     D919 K5
      AND     D9122.9
      ORB
      LD=     D919 K6
      AND     D9123.6
      ORB
      AND     D9124.1
      LD=     D919 K1
      OR=     D919 K2
      AND=    D920 D3020
      ORB
      ANB
      MPS
      AND     T506
      MOV     D9125 D3075
      MPP
      OUT     T506 K10
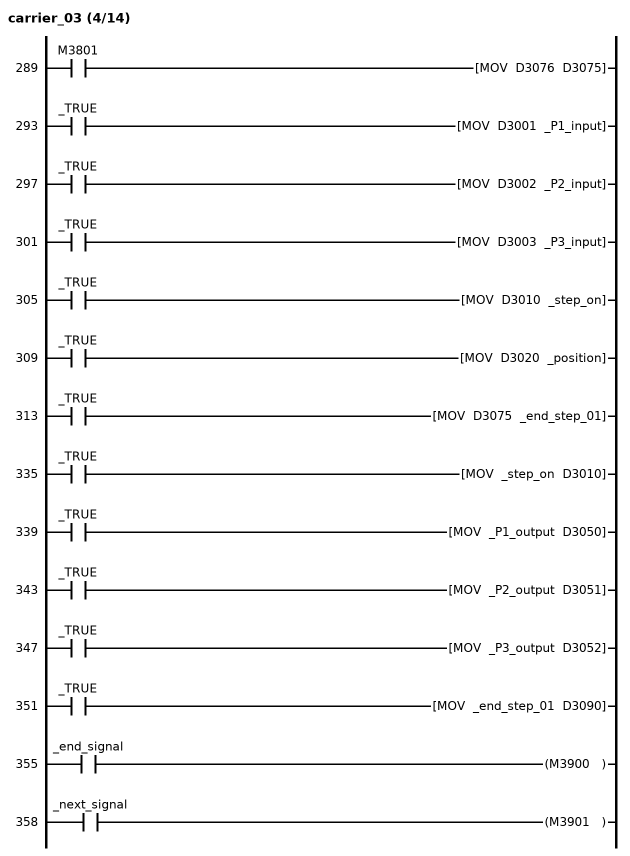
289   LD      M3801
      MOV     D3076 D3075
; FB BLK START c_comm_3(c_comm_3)
293   LD      _TRUE
      MOV     D3001 _P1_input
297   LD      _TRUE
      MOV     D3002 _P2_input
301   LD      _TRUE
      MOV     D3003 _P3_input
305   LD      _TRUE
      MOV     D3010 _step_on
309   LD      _TRUE
      MOV     D3020 _position
313   LD      _TRUE
      MOV     D3075 _end_step_01
; FB START
; FB_NAME c_comm_3
; INSTANCE_NAME c_comm_3
; FB IN_W:P1_input
; FB OUT_step_on:W
; FB IN_W:P2_input
; FB OUT_P1_output:W
; FB IN_W:P3_input
; FB OUT_P2_output:W
; FB IN_W:step_on
; FB OUT_P3_output:W
; FB IN_W:position
; FB OUT_end_step_01:W
; FB IN_W:end_step_01
; FB OUT_end_signal:B
; FB OUT_next_signal:B
; FB OUT_punch:B
; FB END
335   LD      _TRUE
      MOV     _step_on D3010
339   LD      _TRUE
      MOV     _P1_output D3050
343   LD      _TRUE
      MOV     _P2_output D3051
347   LD      _TRUE
      MOV     _P3_output D3052
351   LD      _TRUE
      MOV     _end_step_01 D3090
355   LD      _end_signal
      OUT     M3900
358   LD      _next_signal
      OUT     M3901
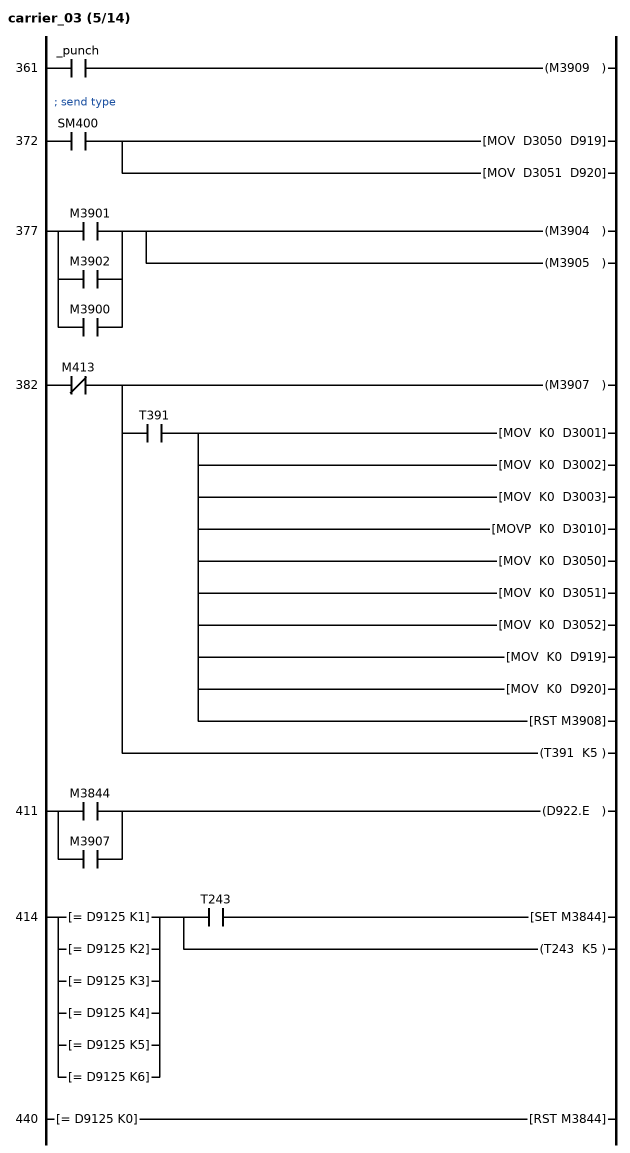
361   LD      _punch
      OUT     M3909
; FB BLK END
; send type
372   LD      SM400
      MOV     D3050 D919
      MOV     D3051 D920
377   LD      M3901
      OR      M3902
      OR      M3900
      OUT     M3904
      OUT     M3905
382   LDI     M413
      OUT     M3907
      MPS
      AND     T391
      MOV     K0 D3001
      MOV     K0 D3002
      MOV     K0 D3003
      MOVP    K0 D3010
      MOV     K0 D3050
      MOV     K0 D3051
      MOV     K0 D3052
      MOV     K0 D919
      MOV     K0 D920
      RST     M3908
      MPP
      OUT     T391 K5
411   LD      M3844
      OR      M3907
      OUT     D922.E
414   LD=     D9125 K1
      OR=     D9125 K2
      OR=     D9125 K3
      OR=     D9125 K4
      OR=     D9125 K5
      OR=     D9125 K6
      MPS
      AND     T243
      SET     M3844
      MPP
      OUT     T243 K5
440   LD=     D9125 K0
      RST     M3844
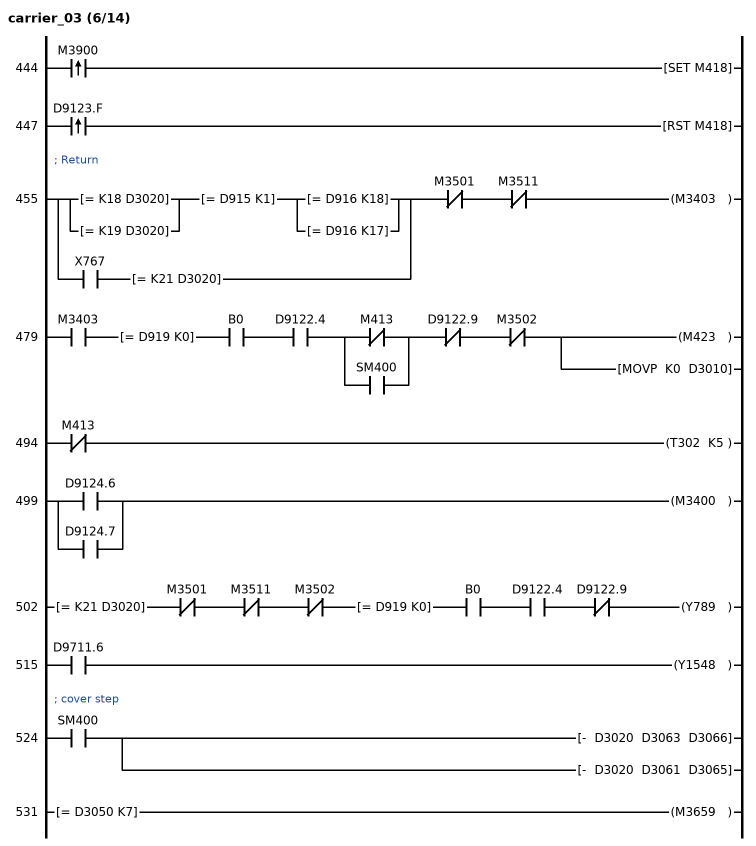
444   LDP     M3900
      SET     M418
447   LDP     D9123.F
      RST     M418
; Return
455   LD=     K18 D3020
      OR=     K19 D3020
      AND=    D915 K1
      LD=     D916 K18
      OR=     D916 K17
      ANB
      LD      X767
      AND=    K21 D3020
      ORB
      ANI     M3501
      ANI     M3511
      OUT     M3403
479   LD      M3403
      AND=    D919 K0
      AND     B0
      AND     D9122.4
      LDI     M413
      OR      SM400
      ANB
      ANI     D9122.9
      ANI     M3502
      OUT     M423
      MOVP    K0 D3010
494   LDI     M413
      OUT     T302 K5
499   LD      D9124.6
      OR      D9124.7
      OUT     M3400
502   LD=     K21 D3020
      ANI     M3501
      ANI     M3511
      ANI     M3502
      AND=    D919 K0
      AND     B0
      AND     D9122.4
      ANI     D9122.9
      OUT     Y789
515   LD      D9711.6
      OUT     Y1548
; cover step
524   LD      SM400
      -       D3020 D3063 D3066
      -       D3020 D3061 D3065
531   LD=     D3050 K7
      OUT     M3659
